// TIA Portal V18 export
TYPE "PLC_TO_KISTLER"
// stored: IsFailsafeCompliant false
   STRUCT
      "0.0" : Bool;   // Start Measure
      "0.1" : Bool;   // Channel Y (Force) Tare Or Reset Piezo
      "0.2" : Bool;   // Channel X (Position) Zero
      "0.3" : Bool;   // Trigger Sensor Test For X
      "0.4" : Bool;   // Trigger Sensor Test For Y
      "0.5" : Bool;   // Reserved
      "0.6" : Bool;   // Master measurement
      "0.7" : Bool;   // Zero incremental sensor
      "1.0" : Bool;   // Reserved
      "1.1" : Bool;   // Acknowledgement With Admin Rights
      "1.2" : Bool;   // Reserved
      "1.3" : Bool;   // Allows PLC To Give The Operator Access Rights
      "1.4" : Bool;   // Bit AUTO, if 1 the PLC has full control over maXYmo
      "1.5" : Bool;   // Reset Statistics
      "1.6" : Bool;   // Deactivate Statistics
      "1.7" : Bool;   // Ext. channel Y Tare or Reset Piezo (MaXYmos NC)
      "2" : Byte;   // Measurement program selection
      "3.0" : Bool;   // Reserved
      "3.1" : Bool;   // Reserved
      "3.2" : Bool;   // Resetting of counter of global serial number
      "3.3" : Bool;   // Reserved
      "3.4" : Bool;   // Reserved
      "3.5" : Bool;   // Reserved
      "3.6" : Bool;   // Reserved
      "3.7" : Bool;   // Reserved
      "4.0" : Bool;   // UNI_0（Freely configurable digital input signal）
      "4.1" : Bool;   // UNI_1
      "4.2" : Bool;   // UNI_2
      "4.3" : Bool;   // UNI_3
      "4.4" : Bool;   // UNI_4
      "4.5" : Bool;   // UNI_5
      "4.6" : Bool;   // UNI_6
      "4.7" : Bool;   // UNI_7
      "5.0" : Bool;   // Reserved
      "5.1" : Bool;   // Reserved
      "5.2" : Bool;   // Reserved
      "5.3" : Bool;   // Reserved
      "5.4" : Bool;   // Reserved
      "5.5" : Bool;   // Reserved
      "5.6" : Bool;   // Reserved
      "5.7" : Bool;   // Reserved
      "6.0" : Bool;   // Reserved
      "6.1" : Bool;   // Reserved
      "6.2" : Bool;   // Reserved
      "6.3" : Bool;   // Reserved
      "6.4" : Bool;   // Reserved
      "6.5" : Bool;   // Reserved
      "6.6" : Bool;   // Reserved
      "6.7" : Bool;   // Reserved
      "7.0" : Bool;   // Reserved
      "7.1" : Bool;   // Reserved
      "7.2" : Bool;   // Reserved
      "7.3" : Bool;   // Reserved
      "7.4" : Bool;   // Reserved
      "7.5" : Bool;   // Reserved
      "7.6" : Bool;   // Reserved
      "7.7" : Bool;   // Reserved
      "8.0" : Bool;   // Reserved
      "8.1" : Bool;   // Reserved
      "8.2" : Bool;   // Reserved
      "8.3" : Bool;   // Reserved
      "8.4" : Bool;   // Reserved
      "8.5" : Bool;   // Reserved
      "8.6" : Bool;   // Reserved
      "8.7" : Bool;   // Reserved
      "9.0" : Bool;   // Enable Drive
      "9.1" : Bool;   // Command Sequence Has Been Run
      "9.2" : Bool;   // Command movement to home position (MP-specific)
      "9.3" : Bool;   // Command movement to reference position (global)
      "9.4" : Bool;   // Command jogging forwards
      "9.5" : Bool;   // Command jogging Backwards
      "9.6" : Bool;   // Continue command sequence after WAIT-REQUEST
      "9.7" : Bool;   // Perform command manual brake test
      "10.0" : Bool;   // Reserved
      "10.1" : Bool;   // Reserved
      "10.2" : Bool;   // Reserved
      "10.3" : Bool;   // External stop sequence
      "10.4" : Bool;   // Reserved
      "10.5" : Bool;   // Reserved
      "10.6" : Bool;   // Reserved
      "10.7" : Bool;   // Reserved
      "11" : Byte;   // Reserved
      "12" : Byte;   // CURRENT SEQUENCE-2
      "13" : Byte;   // Reserved
      "14" : Byte;   // CFG-MP
      "15.0" : Bool;   // Reserved
      "15.1" : Bool;   // Reserved
      "15.2" : Bool;   // Reserved
      "15.3" : Bool;   // Reserved
      "15.4" : Bool;   // Reserved
      "15.5" : Bool;   // Reserved
      "15.6" : Bool;   // Reserved
      "15.7" : Bool;   // Global CFG MP
      "16" : Byte;   // CFG-Address
      "17" : Byte;   // CFG-Lenght
      "18.0" : Bool;   // Select page
      "18.1" : Bool;   // Select page
      "18.2" : Bool;   // Reserved
      "18.3" : Bool;   // Reserved
      "18.4" : Bool;   // Reserved
      "18.5" : Bool;   // Reserved
      "18.6" : Bool;   // Reserved
      "18.7" : Bool;   // Reserved
      "19.0" : Bool;   // Save to MAP
      "19.1" : Bool;   // Strobe
      "19.2" : Bool;
      "19.3" : Bool;
      "19.4" : Bool;   // Changed selected Map
      "19.5" : Bool;
      "19.6" : Bool;   // Changed global
      "19.7" : Bool;   // Backup request
      "20" : Array[1..50] of Char;   // DMC pump
      "70" : Real;   // servoJogSpeed
      "74" : Real;   // ServoManualMaxForce
      EO_01 : Struct
         X_Position_LL : Real;
         X_Position_UL : Real;
         Y_Force_LL : Real;
         Y_Force_UL : Real;
      END_STRUCT;
      EO_02 : Struct
         X_Position_LL : Real;
         X_Position_UL : Real;
         Y_Force_LL : Real;
         Y_Force_UL : Real;
      END_STRUCT;
      EO_03 : Struct
         X_Position_LL : Real;
         X_Position_UL : Real;
         Y_Force_LL : Real;
         Y_Force_UL : Real;
      END_STRUCT;
      EO_04 : Struct
         X_Position_LL : Real;
         X_Position_UL : Real;
         Y_Force_LL : Real;
         Y_Force_UL : Real;
      END_STRUCT;
      EO_05 : Struct
         X_Position_LL : Real;
         X_Position_UL : Real;
         Y_Force_LL : Real;
         Y_Force_UL : Real;
      END_STRUCT;
      EO_06 : Struct
         X_Position_LL : Real;
         X_Position_UL : Real;
         Y_Force_LL : Real;
         Y_Force_UL : Real;
      END_STRUCT;
      "174" : Array[1..46] of Byte;
   END_STRUCT;
END_TYPE
